{region '#Template'}
	{attribute 'Version' := '5.0.0.0'}
	{attribute 'Tags' := '"LCID": "1031", "Text": "DUT, Types, Publisher, Subscriber, AC, General, Settings"'}
	{attribute 'Tags' := '"LCID": "1033", "Text": "DUT, Types, Publisher, Subscriber, AC, General, Settings"'}
	{attribute 'Description' := '"LCID": "1031", "Text": "Basis Daten AC"'}
	{attribute 'Description' := '"LCID": "1033", "Text": "Basic data AC"'}
{endregion}
TYPE ST_BA_GeneralSettings :
STRUCT
	fFrostProtectionSetpoint			: REAL;  // frost protection setpoint. for eg. Heating circutis in protection mode
	fTWth								: REAL;  // present value of outside temperature

	fTWthLowLimit						: REAL;  // below this value all frostprotection funcktions in HVAC-Plants will be enabled
	fTWthDamped							: REAL;  // damped outside temperature

	bTWthLowLimit						: BOOL;  // is TRUE when the outside temperature is below the value from fTWthLmtCrit 
	bTWthDampedLowLimit					: BOOL;  // is TRUE when the damped outside temperature is below the value from fTWthLmtCrit 

	nDummy								: ARRAY [1..6] OF BYTE;
END_STRUCT
END_TYPE

(* stored: Version 1.1.0.1, ProductVersion 3.1.4024.12
   DUT ST_BA_GeneralSettings: Id {13649a3b-4241-4793-8ae7-ff96007c099b} *)
